{attribute 'linkalways'} 
{attribute 'no_explicit_call' := 'This FB is a CLASS and must be accessed using methods or properties'}
{attribute 'enable_dynamic_creation'}
FUNCTION_BLOCK FINAL BooleanDisplayNode EXTENDS Node
VAR
	in : _BOOL(FALSE);
	display : _BOOL(FALSE);
END_VAR

METHOD PUBLIC Clone : I_Node
VAR
	pNode : POINTER TO BooleanDisplayNode;
END_VAR
pNode := __NEW(BooleanDisplayNode);
Clone := pNode^;
END_METHOD

METHOD FB_init : BOOL
VAR_INPUT
	bInitRetains : BOOL; // if TRUE, the retain variables are initialized (warm start / cold start)
	bInCopyCode : BOOL;  // if TRUE, the instance afterwards gets moved into the copy code (online change)
END_VAR
AddInput('in', in);
AddContent('display', display);
END_METHOD

METHOD PROTECTED OnExecute : HRESULT
display.Value := in.Value;
END_METHOD

END_FUNCTION_BLOCK

(* stored: Version 1.1.0.1, ProductVersion 3.1.4024.12
   POU BooleanDisplayNode: Id {de604663-3bb0-00b0-0ba5-dab3958ddc59}, SpecialFunc None
   Folder Constructor: Id {408df8d1-9ce9-4a8b-9803-a2c7e2dccaca}
   Method Clone: Id {39f9c8f2-b07a-4e5c-9803-1cf088bb7713}
   Method FB_init: Id {3a07f333-727b-48f1-94e4-a833a1c151f5}
   Method OnExecute: Id {f90656e7-4e51-03bf-2e02-70618687d7bf} *)
